(* IEC 61131-3 sources: AXOpen/src/templates.simple/ctrl/src, 3 files *)

(* ---- Context.st ---- *)
USING AXOpen.Core;
USING AXOpen.Data;

NAMESPACE axosimple
    CLASS PUBLIC Context EXTENDS AxoContext
        VAR PUBLIC
            ControlledUnit : axosimple.SampleControlledUnit.ControlledUnit;
            ProductionSettings : ProductionSettingsHandler;
            Inputs : REF_TO axosimple.Inputs;
            Outputs : REF_TO axosimple.Outputs;
        END_VAR

        METHOD PROTECTED OVERRIDE Main

            ProductionSettings.Run(THIS);

            IF(Inputs <> NULL AND Outputs <> NULL) THEN
                ControlledUnit.Run(THIS, Inputs^, Outputs^);
            END_IF;
        END_METHOD
    END_CLASS

    CLASS ProductionSettingsHandler EXTENDS AXOpen.Data.AxoDataExchange
        VAR PUBLIC
            {#ix-attr:[AXOpen.Data.DataEntityAttribute]}
            Data : ProductionSettings;
        END_VAR
    END_CLASS

    CLASS ProductionSettings EXTENDS AXOpen.Data.AxoDataEntity
        VAR PUBLIC
            StepDelay : TIME;
        END_VAR

    END_CLASS
END_NAMESPACE

(* ---- configuration.st ---- *)
USING axosimple;
CONFIGURATION MyConfiguration
    TASK Main(Interval := T#10ms, Priority := 1);
    PROGRAM P1 WITH Main: MyProgram;

    VAR_GLOBAL
        Inputs : axosimple.Inputs;
        Outputs : axosimple.Outputs;
        Context : axosimple.Context;
        S71500Rtc :  AXOpen.S71500.Rtc;
        ContextLogger : AXOpen.Messaging.AxoLogger;
    END_VAR
END_CONFIGURATION

(* ---- program.st ---- *)
USING axosimple;
PROGRAM MyProgram
    VAR_EXTERNAL
        Inputs : axosimple.Inputs;
        Outputs : axosimple.Outputs;
        Context : axosimple.Context;
    END_VAR
    // Never modif this the context needs references to IN/OUT structures before it is used.
    Context.Inputs := REF(Inputs);
    Context.Outputs := REF(Outputs);

    // Executes the main context of this application.
    Context.Run();
END_PROGRAM
